INTERFACE ITF_EM_Can_Supply

END_INTERFACE

(* stored: Version 1.1.0.1, ProductVersion 3.1.4024.12
   Itf ITF_EM_Can_Supply: Id {9d641b33-4995-46d9-8141-81fb86fa69d0} *)
